{attribute 'qualified_only'}
(****************** {attribute 'strict'} *)(* Want to treat them as integer constants*)
TYPE ShutterSide :
(
	MINUSX, (* The -X side.*)
    PLUSX   (* The +X side.*)
)INT;
END_TYPE

(* stored: Version 1.1.0.1, ProductVersion 3.1.4020.12
   DUT ShutterSide: Id {e52b5303-1e77-4663-89b3-65730e490f44} *)
